Universal Robots PolyScope program: task_3_lab_3_6_balls_final.urp

Program task_3_lab_3_6_balls_final (installation=default directory=/programs/usbdisk_0/ME5286/Ankush/Lab 3/In Lab/Task 3 createdIn=3.15.8.106339 lastSavedIn=3.15.8.106339 robotSerialNumber=2016352577)
Calibrated DH parameters: a=[0, -0.425, -0.39225, 0, 0, 0]; d=[0.089159, 0, 0, 0.10915, 0.09465, 0.0823]; alpha=[1.570796, 0, 0, 1.570796, -1.570796, 0]; deltaTheta=[0, 0, 0, 0, 0, 0]
Robot Program (runOnlyOnce=true)
  Script file /programs/usbdisk_0/ME5286/Ankush/Lab 3/In Lab/Task 3/Task_3_Lab_3.script
    | def Task3():
    |   # Default parameters:
    |   global speed_ms    = 0.050
    |   global speed_rads  = 0.750
    |   global accel_mss   = 0.100
    |   global accel_radss = 1.200
    |   global blend_radius_m = 0.001
    |   #########################################################
    |   #Chuck Initialization
    |   #########################################################
    |   # define the pins for the chuck
    |   global pin_clamp = 0   # clamp valve digital pin
    |   global pin_unclamp = 2 # unclamp valve digital pin
    |   global pin_objectSense = 0 # photo sensor digital input pin
    | 
    |   # Add any suprograms here
    |   # Main program:
    |   # Program generated by RoboDK v5.6.2 for UR5 on 14/02/2025 11:31:41
    |   # set_reference(p[0.000000, 0.000000, 0.000000, 0.000000, 0.000000, 0.000000])
    |   set_tcp(p[0.000000, 0.000000, 0.211500, 0.000000, 0.000000, 0.000000])
    |   movej([-0.500236, -1.225942, -1.646579, -1.839874, 1.570796, -1.023835],accel_radss,speed_rads,0,0)
    |   rq_set_force(100)
    |   rq_set_speed(100)
    |   speed_ms    = 0.250
    |   accel_mss   = 0.200
    |   # set_reference(p[0.000000, 0.000000, 0.000000, 0.000000, 0.000000, 0.000000])
    |   set_tcp(p[0.000000, 0.000000, 0.211500, 0.000000, 0.000000, 0.000000])
    |   movej([-0.812435, -1.604294, -1.717828, -1.390265, 1.570796, -1.553169],accel_radss,speed_rads,0,blend_radius_m)
    |   speed_ms    = 0.050
    |   accel_mss   = 0.100
    |   # set_reference(p[0.000000, 0.000000, 0.000000, 0.000000, 0.000000, 0.000000])
    |   set_tcp(p[0.000000, 0.000000, 0.211500, 0.000000, 0.000000, 0.000000])
    |   movel(p[0.260567, -0.433543, 0.000000, 2.874883, -1.266749, 0.000000],accel_mss,speed_ms,0,blend_radius_m)
    |   rq_close()
    |   sleep(2)
    |   speed_ms    = 0.050
    |   accel_mss   = 0.100
    |   speed_ms    = 0.050
    |   accel_mss   = 0.100
    |   # set_reference(p[0.000000, 0.000000, 0.000000, 0.000000, 0.000000, 0.000000])
    |   set_tcp(p[0.000000, 0.000000, 0.211500, 0.000000, 0.000000, 0.000000])
    |   movel(p[0.260567, -0.433543, 0.150000, 2.874883, -1.266749, 0.000000],accel_mss,speed_ms,0,blend_radius_m)
    |   speed_ms    = 0.250
    |   accel_mss   = 0.200
    |   # set_reference(p[0.000000, 0.000000, 0.000000, 0.000000, 0.000000, 0.000000])
    |   set_tcp(p[0.000000, 0.000000, 0.211500, 0.000000, 0.000000, 0.000000])
    |   movel(p[0.552361, -0.271266, 0.150000, 2.866767, 1.285010, 0.000000],accel_mss,speed_ms,0,blend_radius_m)
    |   speed_ms    = 0.050
    |   accel_mss   = 0.100
    |   # set_reference(p[0.000000, 0.000000, 0.000000, 0.000000, 0.000000, 0.000000])
    |   set_tcp(p[0.000000, 0.000000, 0.211500, 0.000000, 0.000000, 0.000000])
    |   movel(p[0.552361, -0.271266, 0.000000, 2.866767, 1.285010, 0.000000],accel_mss,speed_ms,0,blend_radius_m)
    |   rq_open()
    |   sleep(2)
    |   speed_ms    = 0.050
    |   accel_mss   = 0.100
    |   # set_reference(p[0.000000, 0.000000, 0.000000, 0.000000, 0.000000, 0.000000])
    |   set_tcp(p[0.000000, 0.000000, 0.211500, 0.000000, 0.000000, 0.000000])
    |   movel(p[0.552361, -0.271266, 0.150000, 2.866767, 1.285010, 0.000000],accel_mss,speed_ms,0,blend_radius_m)
    |   rq_set_force(50)
    |   rq_set_speed(100)
    |   speed_ms    = 0.250
    |   accel_mss   = 0.200
    |   # set_reference(p[0.000000, 0.000000, 0.000000, 0.000000, 0.000000, 0.000000])
    |   set_tcp(p[0.000000, 0.000000, 0.211500, 0.000000, 0.000000, 0.000000])
    |   movej([-0.815441, -1.841567, -1.441199, -1.429627, 1.570796, -1.556176],accel_radss,speed_rads,0,blend_radius_m)
    |   speed_ms    = 0.050
    |   accel_mss   = 0.100
    |   # set_reference(p[0.000000, 0.000000, 0.000000, 0.000000, 0.000000, 0.000000])
    |   set_tcp(p[0.000000, 0.000000, 0.211500, 0.000000, 0.000000, 0.000000])
    |   movel(p[0.329129, -0.508521, 0.000000, 2.874883, -1.266749, 0.000000],accel_mss,speed_ms,0,blend_radius_m)
    |   rq_close()
    |   sleep(2)
    |   speed_ms    = 0.050
    |   accel_mss   = 0.100
    |   speed_ms    = 0.050
    |   accel_mss   = 0.100
    |   # set_reference(p[0.000000, 0.000000, 0.000000, 0.000000, 0.000000, 0.000000])
    |   set_tcp(p[0.000000, 0.000000, 0.211500, 0.000000, 0.000000, 0.000000])
    |   movel(p[0.329129, -0.508521, 0.150000, 2.874883, -1.266749, 0.000000],accel_mss,speed_ms,0,blend_radius_m)
    |   speed_ms    = 0.250
    |   accel_mss   = 0.200
    |   # set_reference(p[0.000000, 0.000000, 0.000000, 0.000000, 0.000000, 0.000000])
    |   set_tcp(p[0.000000, 0.000000, 0.211500, 0.000000, 0.000000, 0.000000])
    |   movel(p[0.619965, -0.195422, 0.150000, 2.866767, 1.285010, 0.000000],accel_mss,speed_ms,0,blend_radius_m)
    |   speed_ms    = 0.050
    |   accel_mss   = 0.100
    |   # set_reference(p[0.000000, 0.000000, 0.000000, 0.000000, 0.000000, 0.000000])
    |   set_tcp(p[0.000000, 0.000000, 0.211500, 0.000000, 0.000000, 0.000000])
    |   movel(p[0.619965, -0.195422, 0.000000, 2.866767, 1.285010, 0.000000],accel_mss,speed_ms,0,blend_radius_m)
    |   rq_open()
    |   sleep(2)
    |   speed_ms    = 0.050
    |   accel_mss   = 0.100
    |   # set_reference(p[0.000000, 0.000000, 0.000000, 0.000000, 0.000000, 0.000000])
    |   set_tcp(p[0.000000, 0.000000, 0.211500, 0.000000, 0.000000, 0.000000])
    |   movel(p[0.619965, -0.195422, 0.150000, 2.866767, 1.285010, 0.000000],accel_mss,speed_ms,0,blend_radius_m)
    |   rq_set_force(100)
    |   rq_set_speed(100)
    |   speed_ms    = 0.250
    |   accel_mss   = 0.200
    |   # set_reference(p[0.000000, 0.000000, 0.000000, 0.000000, 0.000000, 0.000000])
    |   set_tcp(p[0.000000, 0.000000, 0.211500, 0.000000, 0.000000, 0.000000])
    |   movej([-0.694870, -1.462698, -1.853627, -1.396071, 1.570796, -1.435605],accel_radss,speed_rads,0,blend_radius_m)
    |   speed_ms    = 0.050
    |   accel_mss   = 0.100
    |   # set_reference(p[0.000000, 0.000000, 0.000000, 0.000000, 0.000000, 0.000000])
    |   set_tcp(p[0.000000, 0.000000, 0.211500, 0.000000, 0.000000, 0.000000])
    |   movel(p[0.263774, -0.361772, 0.000000, 2.874883, -1.266749, 0.000000],accel_mss,speed_ms,0,blend_radius_m)
    |   rq_close()
    |   sleep(2)
    |   speed_ms    = 0.050
    |   accel_mss   = 0.100
    |   speed_ms    = 0.050
    |   accel_mss   = 0.100
    |   # set_reference(p[0.000000, 0.000000, 0.000000, 0.000000, 0.000000, 0.000000])
    |   set_tcp(p[0.000000, 0.000000, 0.211500, 0.000000, 0.000000, 0.000000])
    |   movel(p[0.263774, -0.361772, 0.150000, 2.874883, -1.266749, 0.000000],accel_mss,speed_ms,0,blend_radius_m)
    |   speed_ms    = 0.250
    |   accel_mss   = 0.200
    |   # set_reference(p[0.000000, 0.000000, 0.000000, 0.000000, 0.000000, 0.000000])
    |   set_tcp(p[0.000000, 0.000000, 0.211500, 0.000000, 0.000000, 0.000000])
    |   movel(p[0.480638, -0.275386, 0.150000, 2.866767, 1.285010, 0.000000],accel_mss,speed_ms,0,blend_radius_m)
    |   speed_ms    = 0.050
    |   accel_mss   = 0.100
    |   # set_reference(p[0.000000, 0.000000, 0.000000, 0.000000, 0.000000, 0.000000])
    |   set_tcp(p[0.000000, 0.000000, 0.211500, 0.000000, 0.000000, 0.000000])
    |   movel(p[0.480638, -0.275386, 0.000000, 2.866767, 1.285010, 0.000000],accel_mss,speed_ms,0,blend_radius_m)
    |   rq_open()
    |   sleep(2)
    |   speed_ms    = 0.050
    |   accel_mss   = 0.100
    |   # set_reference(p[0.000000, 0.000000, 0.000000, 0.000000, 0.000000, 0.000000])
    |   set_tcp(p[0.000000, 0.000000, 0.211500, 0.000000, 0.000000, 0.000000])
    |   movel(p[0.480638, -0.275386, 0.150000, 2.866767, 1.285010, 0.000000],accel_mss,speed_ms,0,blend_radius_m)
    |   rq_set_force(50)
    |   rq_set_speed(100)
    |   speed_ms    = 0.250
    |   accel_mss   = 0.200
    |   # set_reference(p[0.000000, 0.000000, 0.000000, 0.000000, 0.000000, 0.000000])
    |   set_tcp(p[0.000000, 0.000000, 0.211500, 0.000000, 0.000000, 0.000000])
    |   movej([-0.720397, -1.706572, -1.606045, -1.399772, 1.570796, -1.461132],accel_radss,speed_rads,0,blend_radius_m)
    |   speed_ms    = 0.050
    |   accel_mss   = 0.100
    |   # set_reference(p[0.000000, 0.000000, 0.000000, 0.000000, 0.000000, 0.000000])
    |   set_tcp(p[0.000000, 0.000000, 0.211500, 0.000000, 0.000000, 0.000000])
    |   movel(p[0.332337, -0.436751, 0.000000, 2.874883, -1.266749, 0.000000],accel_mss,speed_ms,0,blend_radius_m)
    |   rq_close()
    |   sleep(2)
    |   speed_ms    = 0.050
    |   accel_mss   = 0.100
    |   speed_ms    = 0.050
    |   accel_mss   = 0.100
    |   # set_reference(p[0.000000, 0.000000, 0.000000, 0.000000, 0.000000, 0.000000])
    |   set_tcp(p[0.000000, 0.000000, 0.211500, 0.000000, 0.000000, 0.000000])
    |   movel(p[0.332337, -0.436751, 0.150000, 2.874883, -1.266749, 0.000000],accel_mss,speed_ms,0,blend_radius_m)
    |   speed_ms    = 0.250
    |   accel_mss   = 0.200
    |   # set_reference(p[0.000000, 0.000000, 0.000000, 0.000000, 0.000000, 0.000000])
    |   set_tcp(p[0.000000, 0.000000, 0.211500, 0.000000, 0.000000, 0.000000])
    |   movel(p[0.548241, -0.199542, 0.150000, 2.866767, 1.285010, 0.000000],accel_mss,speed_ms,0,blend_radius_m)
    |   speed_ms    = 0.050
    |   accel_mss   = 0.100
    |   # set_reference(p[0.000000, 0.000000, 0.000000, 0.000000, 0.000000, 0.000000])
    |   set_tcp(p[0.000000, 0.000000, 0.211500, 0.000000, 0.000000, 0.000000])
    |   movel(p[0.548241, -0.199542, 0.000000, 2.866767, 1.285010, 0.000000],accel_mss,speed_ms,0,blend_radius_m)
    |   rq_open()
    |   sleep(2)
    |   speed_ms    = 0.050
    |   accel_mss   = 0.100
    |   # set_reference(p[0.000000, 0.000000, 0.000000, 0.000000, 0.000000, 0.000000])
    |   set_tcp(p[0.000000, 0.000000, 0.211500, 0.000000, 0.000000, 0.000000])
    |   movel(p[0.548241, -0.199542, 0.150000, 2.866767, 1.285010, 0.000000],accel_mss,speed_ms,0,blend_radius_m)
    |   rq_set_force(100)
    |   rq_set_speed(100)
    |   speed_ms    = 0.250
    |   accel_mss   = 0.200
    |   # set_reference(p[0.000000, 0.000000, 0.000000, 0.000000, 0.000000, 0.000000])
    |   set_tcp(p[0.000000, 0.000000, 0.211500, 0.000000, 0.000000, 0.000000])
    |   movej([-0.605727, -1.580184, -1.742507, -1.389696, 1.570796, -1.346462],accel_radss,speed_rads,0,blend_radius_m)
    |   speed_ms    = 0.050
    |   accel_mss   = 0.100
    |   # set_reference(p[0.000000, 0.000000, 0.000000, 0.000000, 0.000000, 0.000000])
    |   set_tcp(p[0.000000, 0.000000, 0.211500, 0.000000, 0.000000, 0.000000])
    |   movel(p[0.335545, -0.364980, 0.000000, 2.874883, -1.266749, 0.000000],accel_mss,speed_ms,0,blend_radius_m)
    |   rq_close()
    |   sleep(2)
    |   speed_ms    = 0.050
    |   accel_mss   = 0.100
    |   speed_ms    = 0.050
    |   accel_mss   = 0.100
    |   # set_reference(p[0.000000, 0.000000, 0.000000, 0.000000, 0.000000, 0.000000])
    |   set_tcp(p[0.000000, 0.000000, 0.211500, 0.000000, 0.000000, 0.000000])
    |   movel(p[0.335545, -0.364980, 0.150000, 2.874883, -1.266749, 0.000000],accel_mss,speed_ms,0,blend_radius_m)
    |   speed_ms    = 0.250
    |   accel_mss   = 0.200
    |   # set_reference(p[0.000000, 0.000000, 0.000000, 0.000000, 0.000000, 0.000000])
    |   set_tcp(p[0.000000, 0.000000, 0.211500, 0.000000, 0.000000, 0.000000])
    |   movel(p[0.476517, -0.203663, 0.150000, 2.866767, 1.285010, 0.000000],accel_mss,speed_ms,0,blend_radius_m)
    |   speed_ms    = 0.050
    |   accel_mss   = 0.100
    |   # set_reference(p[0.000000, 0.000000, 0.000000, 0.000000, 0.000000, 0.000000])
    |   set_tcp(p[0.000000, 0.000000, 0.211500, 0.000000, 0.000000, 0.000000])
    |   movel(p[0.476517, -0.203663, 0.000000, 2.866767, 1.285010, 0.000000],accel_mss,speed_ms,0,blend_radius_m)
    |   rq_open()
    |   sleep(2)
    |   speed_ms    = 0.050
    |   accel_mss   = 0.100
    |   # set_reference(p[0.000000, 0.000000, 0.000000, 0.000000, 0.000000, 0.000000])
    |   set_tcp(p[0.000000, 0.000000, 0.211500, 0.000000, 0.000000, 0.000000])
    |   movel(p[0.476517, -0.203663, 0.150000, 2.866767, 1.285010, 0.000000],accel_mss,speed_ms,0,blend_radius_m)
    |   rq_set_force(50)
    |   rq_set_speed(100)
    |   speed_ms    = 0.250
    |   accel_mss   = 0.200
    |   # set_reference(p[0.000000, 0.000000, 0.000000, 0.000000, 0.000000, 0.000000])
    |   set_tcp(p[0.000000, 0.000000, 0.211500, 0.000000, 0.000000, 0.000000])
    |   movej([-0.644356, -1.821635, -1.466743, -1.424005, 1.570796, -1.385090],accel_radss,speed_rads,0,blend_radius_m)
    |   speed_ms    = 0.050
    |   accel_mss   = 0.100
    |   # set_reference(p[0.000000, 0.000000, 0.000000, 0.000000, 0.000000, 0.000000])
    |   set_tcp(p[0.000000, 0.000000, 0.211500, 0.000000, 0.000000, 0.000000])
    |   movel(p[0.404107, -0.439958, 0.000000, 2.874883, -1.266749, 0.000000],accel_mss,speed_ms,0,blend_radius_m)
    |   rq_close()
    |   sleep(2)
    |   speed_ms    = 0.050
    |   accel_mss   = 0.100
    |   speed_ms    = 0.050
    |   accel_mss   = 0.100
    |   # set_reference(p[0.000000, 0.000000, 0.000000, 0.000000, 0.000000, 0.000000])
    |   set_tcp(p[0.000000, 0.000000, 0.211500, 0.000000, 0.000000, 0.000000])
    |   movel(p[0.404107, -0.439958, 0.150000, 2.874883, -1.266749, 0.000000],accel_mss,speed_ms,0,blend_radius_m)
    |   speed_ms    = 0.250
    |   accel_mss   = 0.200
    |   # set_reference(p[0.000000, 0.000000, 0.000000, 0.000000, 0.000000, 0.000000])
    |   set_tcp(p[0.000000, 0.000000, 0.211500, 0.000000, 0.000000, 0.000000])
    |   movel(p[0.544121, -0.127818, 0.150000, 2.866767, 1.285010, 0.000000],accel_mss,speed_ms,0,blend_radius_m)
    |   speed_ms    = 0.050
    |   accel_mss   = 0.100
    |   # set_reference(p[0.000000, 0.000000, 0.000000, 0.000000, 0.000000, 0.000000])
    |   set_tcp(p[0.000000, 0.000000, 0.211500, 0.000000, 0.000000, 0.000000])
    |   movel(p[0.544121, -0.127818, 0.000000, 2.866767, 1.285010, 0.000000],accel_mss,speed_ms,0,blend_radius_m)
    |   rq_open()
    |   sleep(2)
    |   speed_ms    = 0.050
    |   accel_mss   = 0.100
    |   # set_reference(p[0.000000, 0.000000, 0.000000, 0.000000, 0.000000, 0.000000])
    |   set_tcp(p[0.000000, 0.000000, 0.211500, 0.000000, 0.000000, 0.000000])
    |   movel(p[0.544121, -0.127818, 0.150000, 2.866767, 1.285010, 0.000000],accel_mss,speed_ms,0,blend_radius_m)
    |   # set_reference(p[0.000000, 0.000000, 0.000000, 0.000000, 0.000000, 0.000000])
    |   set_tcp(p[0.000000, 0.000000, 0.211500, 0.000000, 0.000000, 0.000000])
    |   movej([0.000000, -1.570796, 0.000000, -1.570796, 0.000000, 0.000000],accel_radss,speed_rads,0,0)
    |   # End of main program
    | end
    | #####################################################################
    | #closes clamp
    | def clamp():
    | 	if get_standard_digital_in(pin_objectSense):
    | 		#clamp pneumatic clamp
    | 		set_standard_digital_out(pin_clamp, True)
    | 		set_standard_digital_out(pin_unclamp, False)
    | 
    | 		#add a delay in seconds
    | 		sleep(1.0)
    | 
    | 		# Turn the pin off
    | 		set_standard_digital_out(pin_clamp, False)
    | 	else:
    | 		sleep(1.0)
    | 	end
    | end
    | 
    | #####################################################################
    | #opens clamp
    | def unclamp():
    | 	#unclamp pneumatic clamp
    | 	set_standard_digital_out(pin_clamp, False)
    | 	set_standard_digital_out(pin_unclamp, True)
    | 
    | 	#add a delay in seconds
    | 	sleep(1.0)
    | 
    | 	# Turn the pin off
    | 	set_standard_digital_out(pin_unclamp, False)
    | 
    | end
    | 
    | #####################################################################
    | #twist with torque check
    | def tighten_torque(torqueLimit, writst3_StartAngle, wrist3_EndAngle, jointAccel, jointSpeed, num_checkTorque, gripperForce, gripperSpeed, gripperOpen): #In this function, torque limit = max torque to stop turning at, wrist3_StartAngle is angle to start spinning at, wrist3_EndAngle is angle to stop turning at, gripperForce and gripperSpeed are Force and Speed settings of gripper, gripperOpen is how much to open the gripper
    | 	#Get the current joint angle positions
    | 	joint_pos = get_actual_joint_positions()
    | 	#Set jointAngle[5] (wrist3) to startAngle
    | 	joint_pos[5] = writst3_StartAngle
    | 
    | 	global joint_inc = norm(wrist3_EndAngle - writst3_StartAngle) / num_checkTorque
    | 	global q = 0
    | 	global joint_torques = get_joint_torques()
    | 
    | 	#Gripper Settings
    |     	rq_set_speed_norm(gripperForce) #0 - 100
    |     	rq_set_force_norm(gripperSpeed) #0 - 100
    | 
    | 	#screw based on torque
    | 	joint_torques[5] = 0
    | 	while norm(joint_torques[5]) < torqueLimit:
    | 		#Move to beginning turn position
    | 		joint_pos[5] = writst3_StartAngle
    | 		movel(joint_pos, jointAccel, jointSpeed)
    | 		#Close the gripper
    | 		rq_move_and_wait_norm(100)
    | 		q = 0
    | 		while q < num_checkTorque:
    | 			#Move to end of twist
    | 			joint_pos[5] = joint_pos[5] + joint_inc
    | 			movel(joint_pos, jointAccel, jointSpeed)
    | 			#get joint torques
    | 			joint_torques = get_joint_torques()
    | 			if norm(joint_torques[5]) > torqueLimit:
    | 				break
    | 			end
    | 			q = q+1
    | 		end
    | 		#open gripper
    | 		rq_move_and_wait_norm(gripperOpen)
    | 	end
    | end
    | 
    | 
    | Task3()
